PROGRAM Get_QRob_Pos
VAR
	
MC_ReadActualPosition : MC_ReadActualPosition;
actual_position : REAL;

Driver_temperature_C AT%I*:UINT:= 0;


    FB_CoERead_ByDriveRef : FB_CoERead_ByDriveRef;
    stDriveRef        :  ST_DriveRef := (sNetId:= '172.18.236.0.6.1', nDriveNo := 1, nDriveType := 16, nSlaveAddr := 1001); 

    Index             : WORD := 16#22A2;
    SubIndex          : BYTE := 0; 
    Execute           : BOOL := TRUE;
    Timeout           : TIME := T#5S;
    CompleteAccess    : BOOL := TRUE;
    vendorId          : UINT ;
    Error             : BOOL;
    AdsErrId          : UDINT;
    CANopenErrId      : UDINT;
	
	FB_EcCoESdoRead : FB_EcCoESdoRead;
	dir :  T_AmsNetId := '172.18.236.0.6.1';
	
	pSample : POINTER TO UINT;
	driver_temperature : UINT;
	
	Cooler_fan AT%Q*:BOOL:= FALSE;
	Temperature_Ctr : Temperature_Ctr;

END_VAR

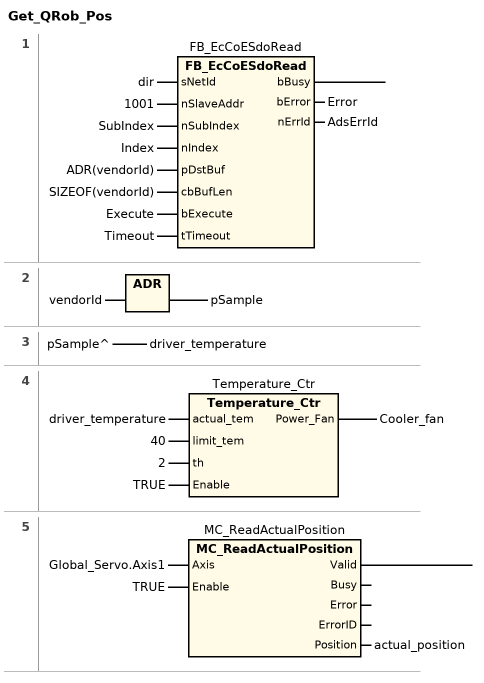
// NETWORK 1
FB_EcCoESdoRead(
    sNetId := dir,
    nSlaveAddr := 1001,
    nSubIndex := SubIndex,
    nIndex := Index,
    pDstBuf := ADR(vendorId),
    cbBufLen := SIZEOF(vendorId),
    bExecute := Execute,
    tTimeout := Timeout,
    bError => Error,
    nErrId => AdsErrId);

// NETWORK 2
pSample := ADR(vendorId);

// NETWORK 3
driver_temperature := pSample^;

// NETWORK 4
Temperature_Ctr(actual_tem := driver_temperature, limit_tem := 40, th := 2, Enable := TRUE);
Cooler_fan := Temperature_Ctr.Power_Fan;

// NETWORK 5
MC_ReadActualPosition(Axis := Global_Servo.Axis1, Enable := TRUE, Position => actual_position);

END_PROGRAM

(* stored: Version 1.1.0.1, ProductVersion 3.1.4024.4
   POU Get_QRob_Pos: Id {6df7057f-e3e5-4f0d-bca7-ae6bdd00b6f3}, SpecialFunc None *)
